FUNCTION_BLOCK FB_Pump EXTENDS StateMachineBase IMPLEMENTS I_HydrualicPump
VAR_INPUT
    bIsSimulator : BOOL;
	bPumpRelay : BOOL; // Option: has pump with relay only
	bPumpHPU : BOOL; // Option: has Hydrualic Power Unit (HPU)
END_VAR
VAR_OUTPUT
END_VAR
VAR
    //fInputSignal : LREAL;
END_VAR

METHOD getSignal : BOOL
VAR_INPUT
END_VAR
END_METHOD

METHOD start : BOOL
VAR_INPUT
END_VAR
nextState := eState_Startup;
END_METHOD

METHOD stop : BOOL
VAR_INPUT
END_VAR
nextState := eState_Stopping;
END_METHOD

END_FUNCTION_BLOCK

(* stored: Version 1.1.0.1, ProductVersion 3.1.4024.9
   POU FB_Pump: Id {c4f79673-c352-48af-9b2c-c649dc4f25ab}, SpecialFunc None
   Method getSignal: Id {4b31f716-6658-43ef-a156-6de609a15d27}
   Method start: Id {85ca6983-27bb-4c44-9760-8f51e66523f4}
   Method stop: Id {8ac0dd21-6534-45b4-911c-e5607e880992} *)
